(* CODESYS project OOP example Methods Properties.project

Project tree, tasks and I/O mapping:
  Device : CODESYS Control for Raspberry Pi SL, 3S - Smart Software Solutions GmbH, version 3.5.12.30
    application Application
      libraries: Standard, * (System); VisuDialogs, * (System); SysFile, 3.5.9.0 (System); AlarmManager, 3.5.12.0 (Intern)
      task MainTask (cyclic, interval 500 ms, priority 1, watchdog 1000 ms x 1) calls Methods_Properties
      program Methods_Properties [ST]
    SoftMotion General Axis Pool
    I²C
    SPI
    GPIOs_A_B : GPIOs B+/Pi2, 3S - Smart Software Solutions GmbH, version 3.5.11.0
        unmapped channels: digital inputs (GPIO0..GPIO31), digital outputs (GPIO0..GPIO31)
    Onewire
    Camera device
      <Empty>
  libraries: VisuSymbols, 3.5.10.0 (System)
  Methods & Properties/
    function block FB_Engine [ST]: Start, Stop, MaxVelocity, Temperature, Velocity
*)

// Device/Application/Methods_Properties
PROGRAM Methods_Properties
VAR
	fbEngine : FB_ENGINE;
	temperature : REAL;
    start : BOOL := TRUE;
    rMaxVelocity : REAL := 130; //kmph
    rVelocity : REAL := 100; //kmph
    iGear : INT  := 5;
    xStarted : BOOL;
	xStopped : BOOL;
END_VAR

IF start THEN
    xStarted := fbEngine.Start( iGear:= iGear, rVelocity := rVelocity );
	xStopped := FALSE;
ELSE        
	xStarted := FALSE;
	xStopped 		 := fbEngine.Stop(); 
END_IF

fbEngine.MaxVelocity := rMaxVelocity;
temperature := fbEngine.Temperature; 

// toggle start;
start := NOT start;

END_PROGRAM

// Methods & Properties/FB_Engine
// Class FB_Engine
FUNCTION_BLOCK FB_Engine
VAR
   _xStarted : BOOL;
   _rVelocity : REAL;
   _rMaxVelocity : REAL;
   _iGear : INT;
   _rTemperature : REAL;
END_VAR

//The THIS pointer is available to all function blocks and points to the current function block instance. 
//It is required whenever a method contains a local variable which obscures a variable in the function block.
//
//An assignment statement within the method sets the value of the local variable. 
//If we want the method to set the value of the local variable in the function block, we need to use the THIS pointer to access it.
METHOD Start : Bool;
VAR_INPUT
   rVelocity : REAL;
   iGear     : INT;
END_VAR
THIS^._xStarted  := TRUE;
Start            := TRUE;
THIS^._iGear     := iGear;
THIS^._rVelocity := MIN( ABS(THIS^._rMaxVelocity), rVelocity );

CASE TO_INT( THIS^._rVelocity ) OF // implicit typecasting(TO_INT), use REAL_TO_INT for explicit typecasting
   0..100 :
      THIS^._rTemperature := 50;
   101..1000:
      THIS^._rTemperature := 90;
   1001..10000:
      THIS^._rTemperature := 100;
   10001..32767:
      THIS^._rTemperature := 150;
END_CASE
END_METHOD

METHOD Stop : BOOL
VAR_INPUT
END_VAR
THIS^._xStarted := FALSE;
Stop            := TRUE;
END_METHOD

PROPERTY MaxVelocity : REAL
SET
THIS^._rMaxVelocity := MaxVelocity;
END_SET
GET
MaxVelocity := THIS^._rMaxVelocity;
END_GET
END_PROPERTY

PROPERTY Temperature : REAL
GET
Temperature := THIS^._rTemperature;
END_GET
END_PROPERTY

PROPERTY Velocity : real
GET
Velocity := THIS^._rVelocity;
END_GET
END_PROPERTY

END_FUNCTION_BLOCK
